(* CODESYS project Plc Uppgift 12.project

Project tree, tasks and I/O mapping:
  Device : CODESYS Control Win V3, 3S - Smart Software Solutions GmbH, order no. 305021, version 3.5.10.40
    application Application
      libraries: Standard, * (System)
      task MainTask (cyclic, interval t#20ms, priority 1) calls PLC_PRG
      program PLC_PRG [ST]
      global variables GVL
      Symbols
*)

// Device/Application/GVL
{attribute 'qualified_only'}
VAR_GLOBAL
	Sensor1 : BOOL;
	Sensor2 : BOOL;
	Sensor3 : BOOL;
	Sensor4 : BOOL;
	Sensor5 : BOOL;
	Sensor6 : BOOL;
	Sensor7 : BOOL;
	
	MotorControl1 : BOOL;
	MotorControl2 : BOOL;
	MotorControl3 : BOOL;
	MotorControl4 : BOOL;
	
	TurnControlFwd : BOOL;
	TurnControlRev : BOOL;
	
	DropBox: BOOL;
END_VAR

// Device/Application/PLC_PRG
PROGRAM PLC_PRG
VAR
state: INT; //The main state of the system.
HoldConver2Timmer: TON; // For conveyor 2 to hold for detection.
END_VAR

//Inital start function
//state := 0;

CASE state OF
	// Statestart. - Box detect
	0:
		IF gvl.Sensor6 THEN
			state := 5;
		END_IF
		
		IF gvl.Sensor1 THEN
				state := 1;
		END_IF
	
	// Load box from startpos to moving conveyor.
	1:
		IF gvl.Sensor7 THEN
			IF gvl.Sensor1 THEN
				gvl.MotorControl1 := TRUE;
				gvl.MotorControl2 := TRUE;
			END_IF
		ELSE
			state := 5;
		END_IF
		
		
		IF gvl.Sensor2 THEN
			gvl.MotorControl1 := FALSE;
			gvl.MotorControl2 := FALSE;
			state := 2;
		END_IF

	// end of case 1
	// Detect BOX SIZE.
	2:
		HoldConver2Timmer(IN:= TRUE,PT:= T#1S);
		
		IF HoldConver2Timmer.Q THEN
			IF gvl.Sensor5 THEN
				state := 4;
			ELSE
				state := 3;
			END_IF
			
		END_IF
	
	// end of case 2	
	// Move to conveor 3.
	3:
		IF gvl.Sensor2 THEN
			gvl.MotorControl2 := TRUE;
			gvl.MotorControl3 := TRUE;
		END_IF
		
		IF gvl.Sensor3 THEN
				gvl.MotorControl2 := FALSE;
				gvl.MotorControl3 := FALSE;
				state := 0;
		END_IF
	
	// end of case 3	
	// Move to conveor 4.
	4:
		IF gvl.Sensor7 THEN
			gvl.TurnControlFwd := TRUE;
		END_IF
		
		IF gvl.Sensor6 THEN
			gvl.TurnControlFwd := false;
				gvl.MotorControl2 := TRUE;
				gvl.MotorControl4 := TRUE;
		END_IF
	
		IF gvl.Sensor4 THEN
				gvl.MotorControl2 := FALSE;
				gvl.MotorControl4 := FALSE;
				state := 5;
		END_IF
	// end of case 4
	// Resseting Moving conveor to default place.
	5:
		IF gvl.Sensor6 THEN
			gvl.TurnControlRev := TRUE;
		END_IF
		
		IF gvl.Sensor7 THEN
			gvl.TurnControlRev := FALSE;
			IF gvl.Sensor2 THEN
				state := 2;
			ELSE
				state := 0;
			END_IF
		END_IF
		
	// end of case 5
	ELSE
		state := 0;	
END_CASE

END_PROGRAM
